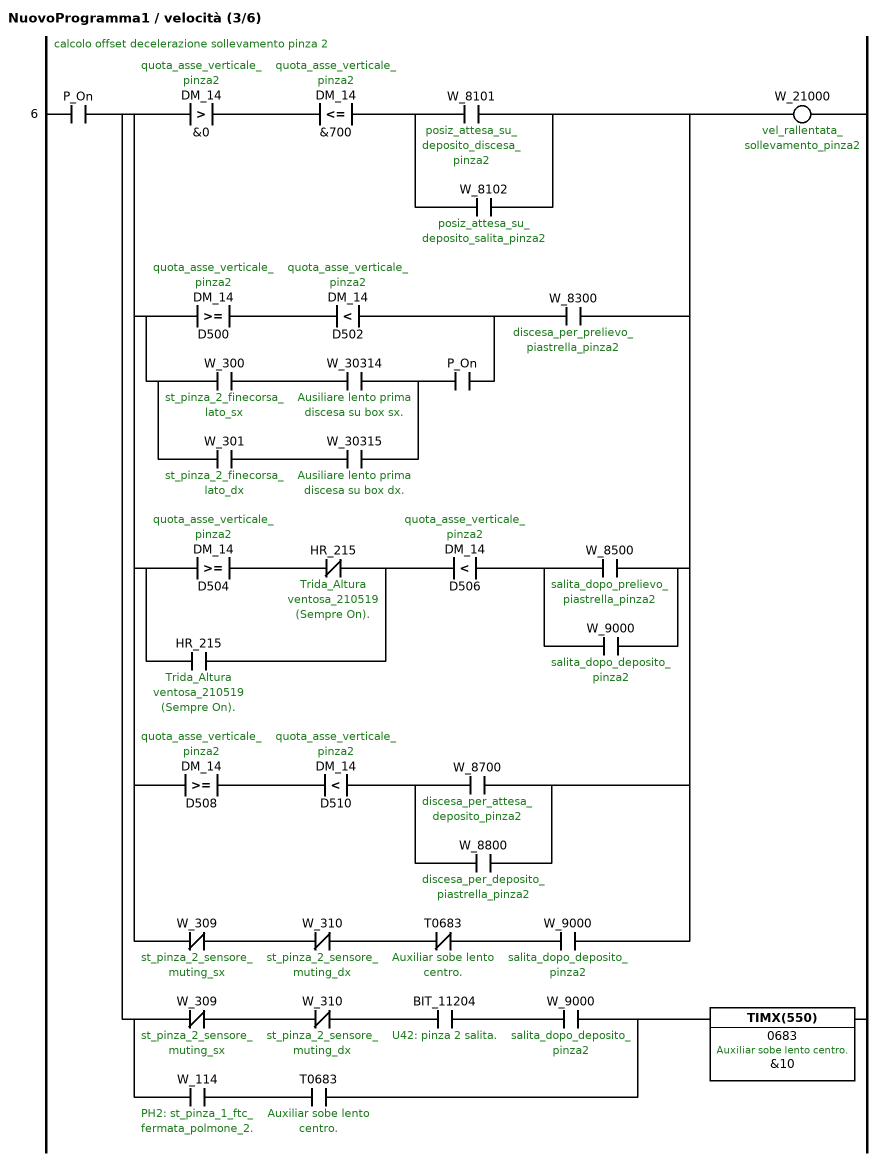
; [picture p120: NuovoProgramma1 / velocità, rungs 6-6]
; rung 6: calcolo offset decelerazione sollevamento pinza 2
LD P_On
OUT TR0
LD>SL(323) DM_14 &0  ; quota_asse_verticale_pinza2
AND<=SL(318) DM_14 &700  ; quota_asse_verticale_pinza2
LD W_8101  ; posiz_attesa_su_deposito_discesa_pinza2
OR W_8102  ; posiz_attesa_su_deposito_salita_pinza2
ANDLD
LD>=SL(328) DM_14 D500  ; quota_asse_verticale_pinza2
AND<SL(313) DM_14 D502  ; quota_asse_verticale_pinza2
LD W_300  ; st_pinza_2_finecorsa_lato_sx
AND W_30314  ; Ausiliare lento prima discesa su box sx.
LD W_301  ; st_pinza_2_finecorsa_lato_dx
AND W_30315  ; Ausiliare lento prima discesa su box dx.
ORLD
AND P_On
ORLD
AND W_8300  ; discesa_per_prelievo_piastrella_pinza2
ORLD
LD>=SL(328) DM_14 D504  ; quota_asse_verticale_pinza2
ANDNOT HR_215  ; Trida_Altura ventosa_210519 (Sempre On).  // HR 2.15: Ventosa voltava a entrar veloz pouco antes de para no alto. / .
OR HR_215  ; Trida_Altura ventosa_210519 (Sempre On).  // HR 2.15: Ventosa voltava a entrar veloz pouco antes de para no alto. / .
AND<SL(313) DM_14 D506  ; quota_asse_verticale_pinza2
LD W_8500  ; salita_dopo_prelievo_piastrella_pinza2
OR W_9000  ; salita_dopo_deposito_pinza2
ANDLD
ORLD
LD>=SL(328) DM_14 D508  ; quota_asse_verticale_pinza2
AND<SL(313) DM_14 D510  ; quota_asse_verticale_pinza2
LD W_8700  ; discesa_per_attesa_deposito_pinza2
OR W_8800  ; discesa_per_deposito_piastrella_pinza2
ANDLD
ORLD
LDNOT W_309  ; st_pinza_2_sensore_muting_sx  // Pinça no centro. / .
ANDNOT W_310  ; st_pinza_2_sensore_muting_dx  // Pinça no centro. / .
ANDNOT T0683  ; Auxiliar sobe lento centro.
AND W_9000  ; salita_dopo_deposito_pinza2
ORLD
ANDLD
OUT W_21000  ; vel_rallentata_sollevamento_pinza2
LD TR0
LDNOT W_309  ; st_pinza_2_sensore_muting_sx  // Pinça no centro. / .
ANDNOT W_310  ; st_pinza_2_sensore_muting_dx  // Pinça no centro. / .
AND BIT_11204  ; U42: pinza 2 salita.
AND W_9000  ; salita_dopo_deposito_pinza2
LD W_114  ; PH2: st_pinza_1_ftc_fermata_polmone_2.
AND T0683  ; Auxiliar sobe lento centro.  // Auto-alimento para efetuar controle de velocidade somente no 1º plano depositado. / .
ORLD
ANDLD
TIMX(550) 0683 &10  ; Auxiliar sobe lento centro.  // Auxiliar início sobe lento centro. / "Puxa" as peças do 1º plano depositado. / .

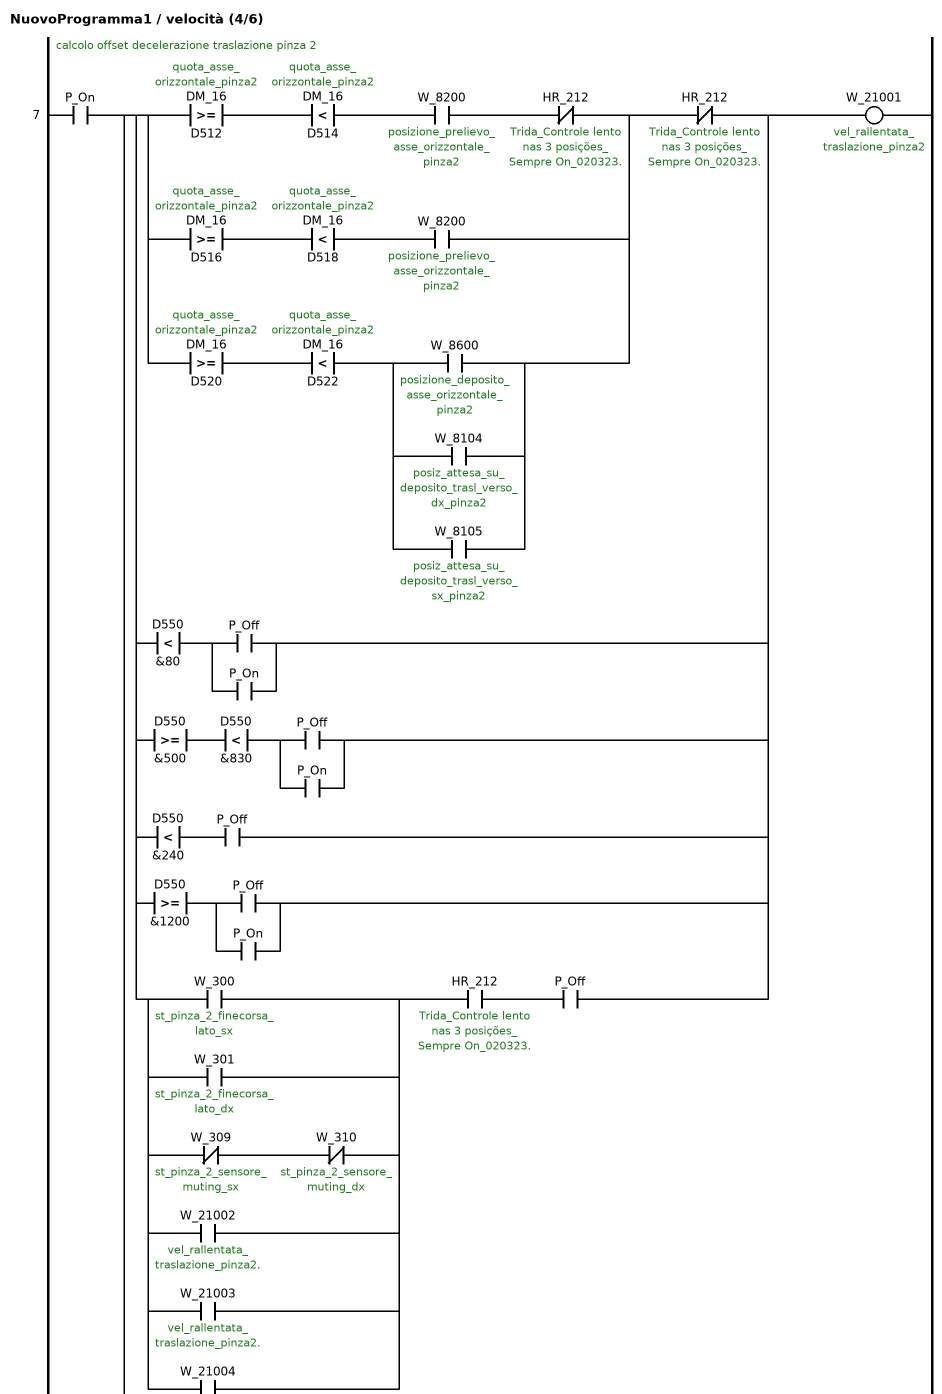

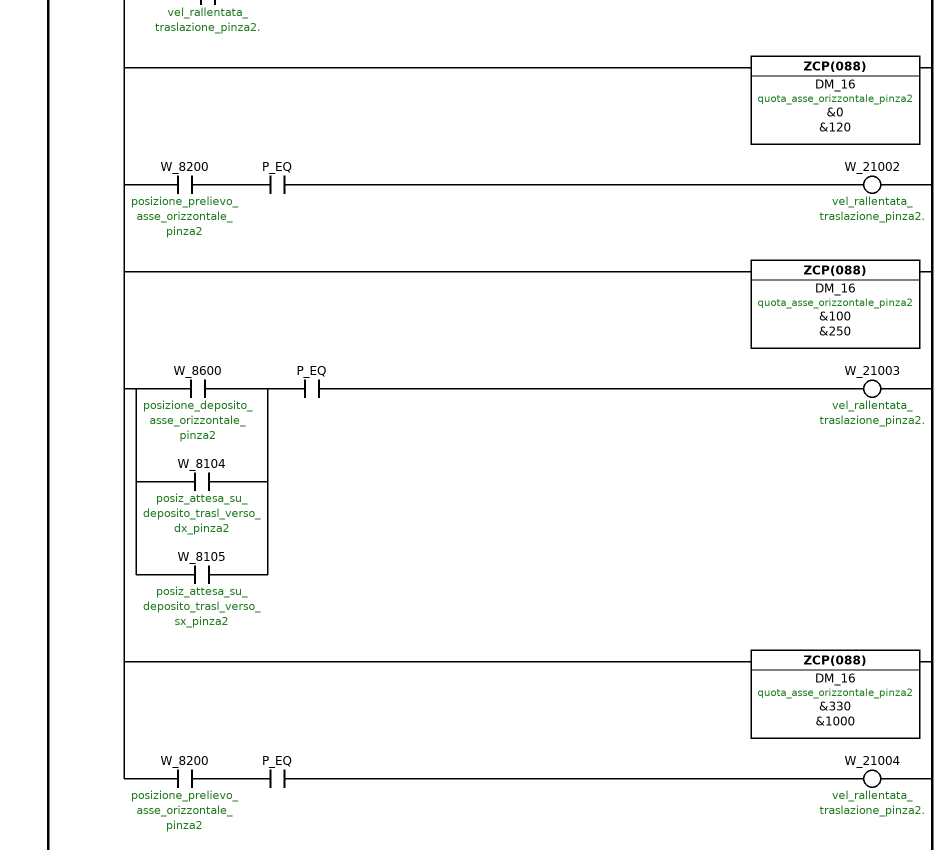
; rung 7: calcolo offset decelerazione traslazione pinza 2
LD P_On
OUT TR0
LD>=SL(328) DM_16 D512  ; quota_asse_orizzontale_pinza2
AND<SL(313) DM_16 D514  ; quota_asse_orizzontale_pinza2
AND W_8200  ; posizione_prelievo_asse_orizzontale_pinza2
ANDNOT HR_212  ; Trida_Controle lento nas 3 posições_Sempre On_020323.
LD>=SL(328) DM_16 D516  ; quota_asse_orizzontale_pinza2
AND<SL(313) DM_16 D518  ; quota_asse_orizzontale_pinza2
AND W_8200  ; posizione_prelievo_asse_orizzontale_pinza2
ORLD
LD>=SL(328) DM_16 D520  ; quota_asse_orizzontale_pinza2
AND<SL(313) DM_16 D522  ; quota_asse_orizzontale_pinza2
LD W_8600  ; posizione_deposito_asse_orizzontale_pinza2
OR W_8104  ; posiz_attesa_su_deposito_trasl_verso_dx_pinza2
OR W_8105  ; posiz_attesa_su_deposito_trasl_verso_sx_pinza2
ANDLD
ORLD
ANDNOT HR_212  ; Trida_Controle lento nas 3 posições_Sempre On_020323.
LD<SL(313) D550 &80
LD P_Off
OR P_On
ANDLD
ORLD
LD>=SL(328) D550 &500
AND<SL(313) D550 &830
LD P_Off
OR P_On
ANDLD
ORLD
LD<SL(313) D550 &240
AND P_Off
ORLD
LD>=SL(328) D550 &1200
LD P_Off
OR P_On
ANDLD
ORLD
LD W_300  ; st_pinza_2_finecorsa_lato_sx  // Pinça à esquerda. / .
OR W_301  ; st_pinza_2_finecorsa_lato_dx  // Pinça à direita. / .
LDNOT W_309  ; st_pinza_2_sensore_muting_sx  // Pinça no centro. / .
ANDNOT W_310  ; st_pinza_2_sensore_muting_dx  // Pinça no centro. / .
ORLD
OR W_21002  ; vel_rallentata_traslazione_pinza2.
OR W_21003  ; vel_rallentata_traslazione_pinza2.
OR W_21004  ; vel_rallentata_traslazione_pinza2.
AND HR_212  ; Trida_Controle lento nas 3 posições_Sempre On_020323.
AND P_Off
ORLD
ANDLD
OUT W_21001  ; vel_rallentata_traslazione_pinza2
LD TR0
ZCP(088) DM_16 &0 &120  ; quota_asse_orizzontale_pinza2  // Valor contagem na esquerda: 0. / .
AND W_8200  ; posizione_prelievo_asse_orizzontale_pinza2
AND P_EQ
OUT W_21002  ; vel_rallentata_traslazione_pinza2.
LD TR0
ZCP(088) DM_16 &100 &250  ; quota_asse_orizzontale_pinza2  // Valor contagem no centro: +/- 220. / .
LD W_8600  ; posizione_deposito_asse_orizzontale_pinza2
OR W_8104  ; posiz_attesa_su_deposito_trasl_verso_dx_pinza2
OR W_8105  ; posiz_attesa_su_deposito_trasl_verso_sx_pinza2
ANDLD
AND P_EQ
OUT W_21003  ; vel_rallentata_traslazione_pinza2.
LD TR0
ZCP(088) DM_16 &330 &1000  ; quota_asse_orizzontale_pinza2  // Valor contagem na direita: +/- 360. / .
AND W_8200  ; posizione_prelievo_asse_orizzontale_pinza2
AND P_EQ
OUT W_21004  ; vel_rallentata_traslazione_pinza2.

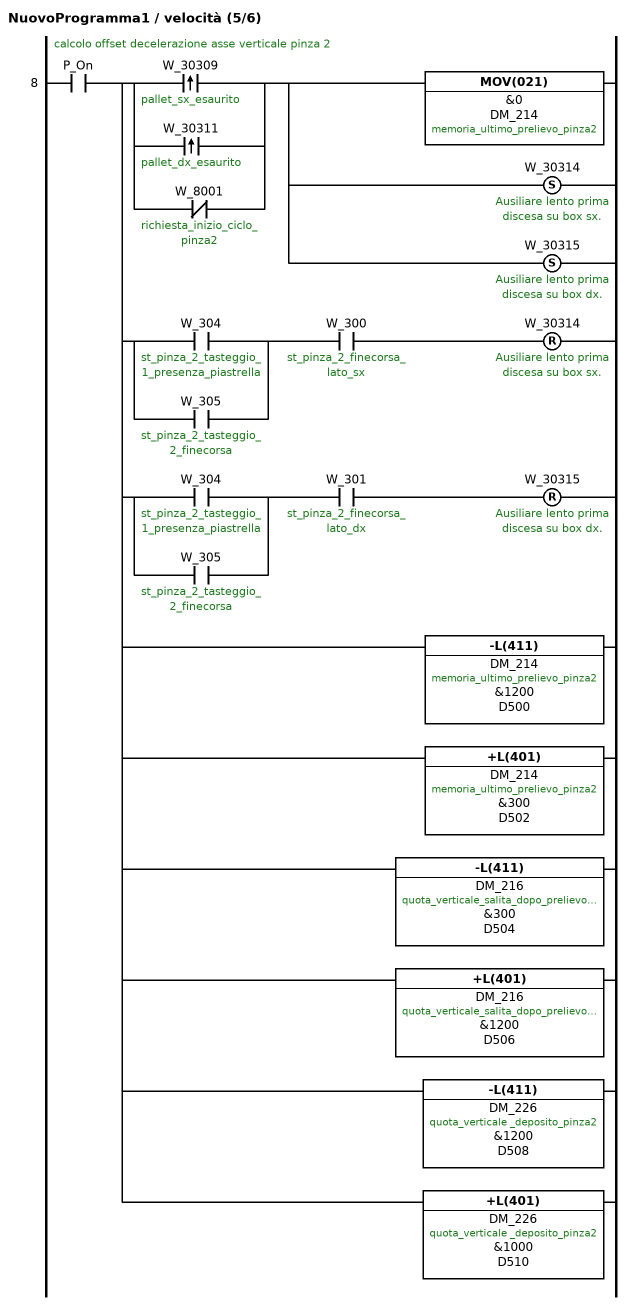
; rung 8: calcolo offset decelerazione asse verticale pinza 2
LD P_On
OUT TR0
@LD W_30309  ; pallet_sx_esaurito
@OR W_30311  ; pallet_dx_esaurito
ORNOT W_8001  ; richiesta_inizio_ciclo_pinza2
ANDLD
MOV(021) &0 DM_214  ; memoria_ultimo_prelievo_pinza2
SET W_30314  ; Ausiliare lento prima discesa su box sx.
SET W_30315  ; Ausiliare lento prima discesa su box dx.
LD TR0
LD W_304  ; st_pinza_2_tasteggio_1_presenza_piastrella
OR W_305  ; st_pinza_2_tasteggio_2_finecorsa
ANDLD
AND W_300  ; st_pinza_2_finecorsa_lato_sx
RSET W_30314  ; Ausiliare lento prima discesa su box sx.
LD TR0
LD W_304  ; st_pinza_2_tasteggio_1_presenza_piastrella
OR W_305  ; st_pinza_2_tasteggio_2_finecorsa
ANDLD
AND W_301  ; st_pinza_2_finecorsa_lato_dx
RSET W_30315  ; Ausiliare lento prima discesa su box dx.
LD TR0
-L(411) DM_214 &1200 D500  ; memoria_ultimo_prelievo_pinza2
+L(401) DM_214 &300 D502  ; memoria_ultimo_prelievo_pinza2
-L(411) DM_216 &300 D504  ; quota_verticale_salita_dopo_prelievo_pinza2
+L(401) DM_216 &1200 D506  ; quota_verticale_salita_dopo_prelievo_pinza2
-L(411) DM_226 &1200 D508  ; quota_verticale _deposito_pinza2
+L(401) DM_226 &1000 D510  ; quota_verticale _deposito_pinza2

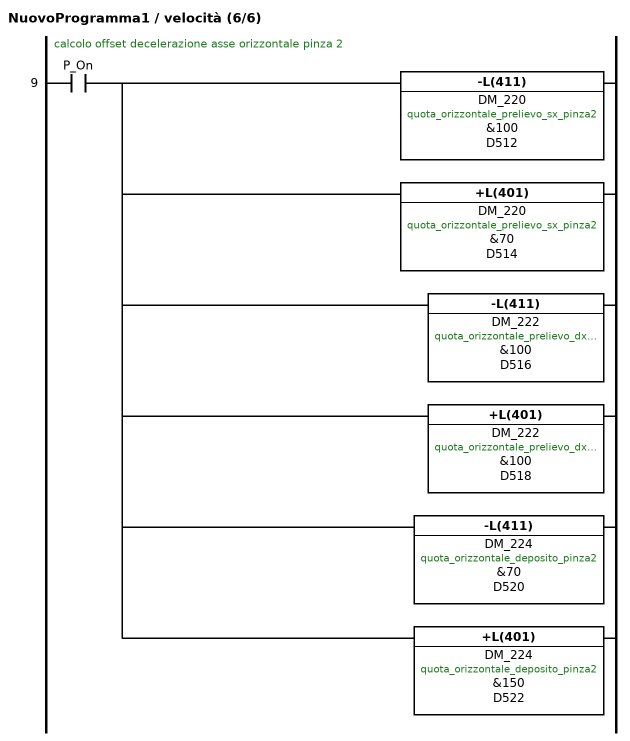
; rung 9: calcolo offset decelerazione asse orizzontale pinza 2
LD P_On
-L(411) DM_220 &100 D512  ; quota_orizzontale_prelievo_sx_pinza2
+L(401) DM_220 &70 D514  ; quota_orizzontale_prelievo_sx_pinza2
-L(411) DM_222 &100 D516  ; quota_orizzontale_prelievo_dx_pinza2
+L(401) DM_222 &100 D518  ; quota_orizzontale_prelievo_dx_pinza2
-L(411) DM_224 &70 D520  ; quota_orizzontale_deposito_pinza2
+L(401) DM_224 &150 D522  ; quota_orizzontale_deposito_pinza2

### Section END
; rung 0
END(001)

## Program NuovoProgramma2 (interrupt task 140)

### Section Sezione1

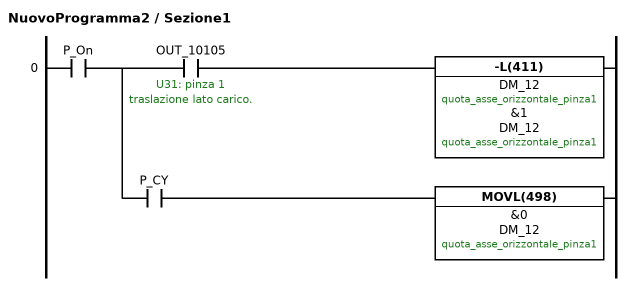
; rung 0
LD P_On
OUT TR0
AND OUT_10105  ; U31: pinza 1 traslazione lato carico.
-L(411) DM_12 &1 DM_12  ; quota_asse_orizzontale_pinza1
LD TR0
AND P_CY
MOVL(498) &0 DM_12  ; quota_asse_orizzontale_pinza1

### Section END
; rung 0
END(001)

## Program NuovoProgramma3 (interrupt task 141)

### Section Sezione1

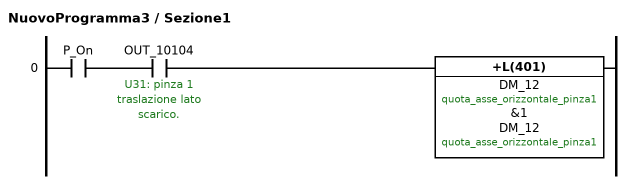
; rung 0
LD P_On
AND OUT_10104  ; U31: pinza 1 traslazione lato scarico.
+L(401) DM_12 &1 DM_12  ; quota_asse_orizzontale_pinza1

### Section END
; rung 0
END(001)

## Program NuovoProgramma4 (interrupt task 142)

### Section Sezione1

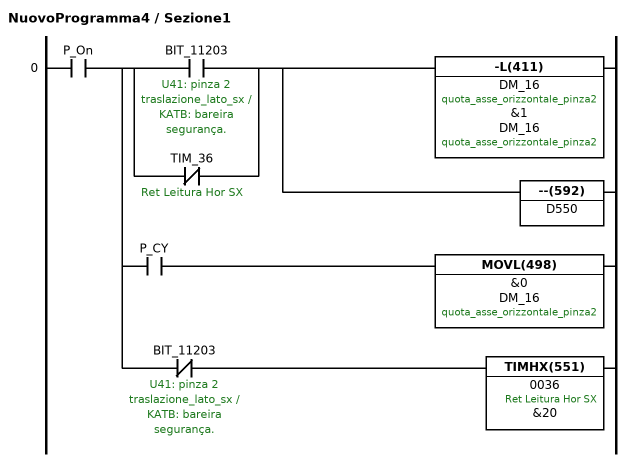
; rung 0
LD P_On
OUT TR0
LD BIT_11203  ; U41: pinza 2 traslazione_lato_sx / KATB: bareira segurança.
ORNOT TIM_36  ; Ret Leitura Hor SX
ANDLD
-L(411) DM_16 &1 DM_16  ; quota_asse_orizzontale_pinza2
--(592) D550
LD TR0
AND P_CY
MOVL(498) &0 DM_16  ; quota_asse_orizzontale_pinza2
LD TR0
ANDNOT BIT_11203  ; U41: pinza 2 traslazione_lato_sx / KATB: bareira segurança.
TIMHX(551) 0036 &20  ; Ret Leitura Hor SX

### Section END
; rung 0
END(001)

## Program NuovoProgramma5 (interrupt task 143)

### Section Sezione1

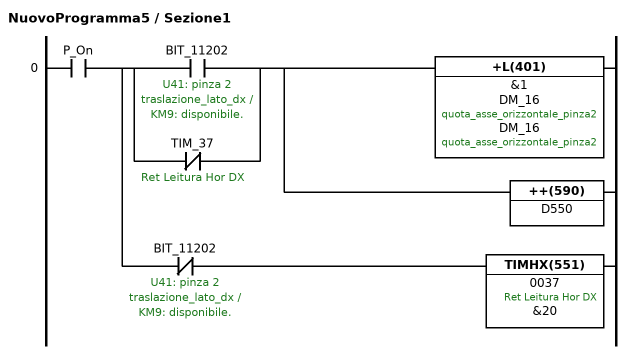
; rung 0
LD P_On
OUT TR0
LD BIT_11202  ; U41: pinza 2 traslazione_lato_dx / KM9: disponibile.
ORNOT TIM_37  ; Ret Leitura Hor DX
ANDLD
+L(401) &1 DM_16 DM_16  ; quota_asse_orizzontale_pinza2
++(590) D550
LD TR0
ANDNOT BIT_11202  ; U41: pinza 2 traslazione_lato_dx / KM9: disponibile.
TIMHX(551) 0037 &20  ; Ret Leitura Hor DX

### Section END
; rung 0
END(001)

## Function block Modbus_Write_Parameter
VAR_INPUT
  Unit_n : INT;
  Serial_port_n : INT;
  Node : INT;
  Parameter : WORD;
  Value : WORD;
  start_comm : BOOL;
END_VAR
VAR_OUTPUT
  Busy : BOOL;
  Comms_error : BOOL;
  Error_Code : WORD;
END_VAR
VAR
  source : ARRAY[0..5] OF WORD;  (* Source area of the CMND *)
  control : ARRAY[0..5] OF WORD;  (* Control Data for the CMND instruction *)
  response : ARRAY[0..4] OF WORD;  (* Response area of the CMND istruction *)
  comm : BOOL;  (* Communication enabled *)
  stop_comm : BOOL;  (* Stops the communication *)
  tmp : DINT;  (* Temporary data for math *)
  port_n AT A218 : WORD;  (* Communication port number assigned with automatic allocation *)
  used_port : WORD;  (* Current communication port *)
  stby : BOOL;  (* Delays the reading of the status for one scan after comms activation *)
  First_Cycle_after_Network_Comms AT A214 : WORD;  (* Turns On on the first scan right after the completion of the communication function *)
  Fisrt_Cycle_after_Comms_Error AT A215 : WORD;  (* Turns On during the first scan after a communication error *)
  error_code_storage_location AT A216 : DWORD;  (* Returns the memory address where the error code is stored *)
  tmp_ir0 : DWORD;  (* Stores the content of IR0 *)
  actual_error_code_ptr : DWORD;  (* Points to the memory location that contains the error code *)
END_VAR

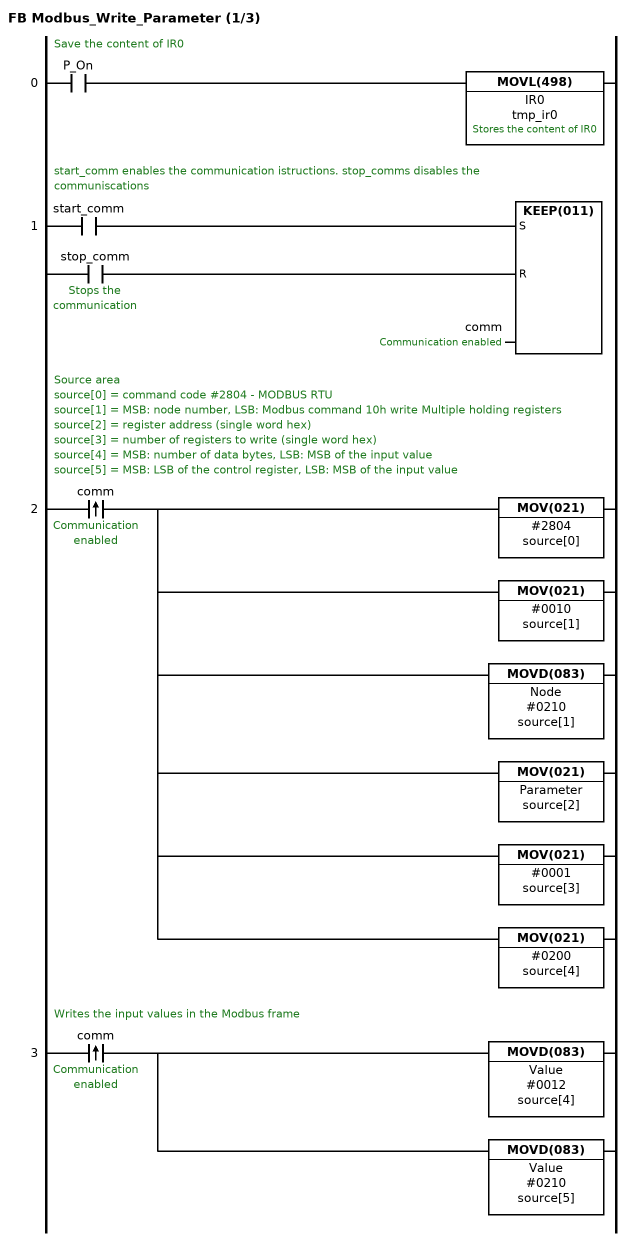
; rung 0: Save the content of IR0
LD P_On
MOVL(498) IR0 tmp_ir0  ; Stores the content of IR0
; rung 1: start_comm enables the communication istructions. stop_comms disables the communiscations
LD start_comm
LD stop_comm  ; Stops the communication
KEEP(011) comm  ; Communication enabled
; rung 2: Source area / source[0] = command code #2804 - MODBUS RTU / source[1] = MSB: node number, LSB: Modbus command 10h write Multiple holding registers / source[2] = register address (single word hex) / source[3] = number of registers to write (single word hex) / source[4] = MSB: number of data bytes, LSB: MSB of the input value / source[5] = MSB: LSB of the control register, LSB: MSB of the input value
@LD comm  ; Communication enabled
MOV(021) #2804 source[0]
MOV(021) #0010 source[1]
MOVD(083) Node #0210 source[1]
MOV(021) Parameter source[2]
MOV(021) #0001 source[3]
MOV(021) #0200 source[4]
; rung 3: Writes the input values in the Modbus frame
@LD comm  ; Communication enabled
MOVD(083) Value #0012 source[4]
MOVD(083) Value #0210 source[5]

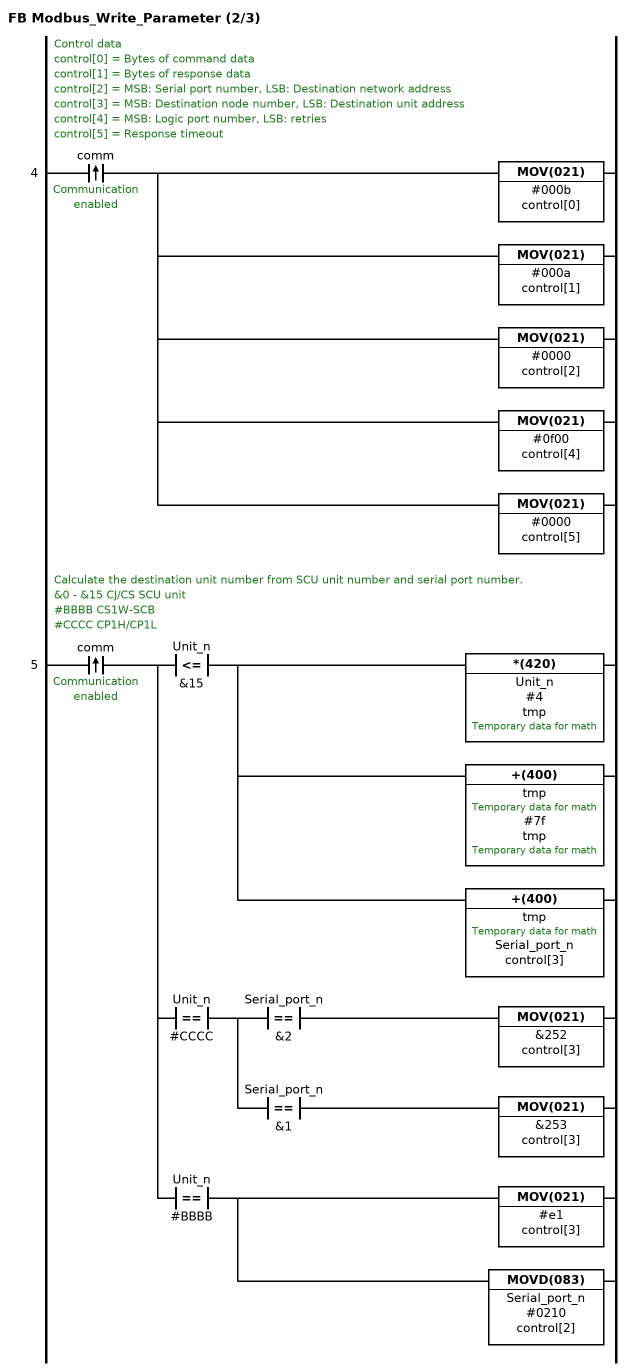
; rung 4: Control data / control[0] = Bytes of command data / control[1] = Bytes of response data / control[2] = MSB: Serial port number, LSB: Destination network address / control[3] = MSB: Destination node number, LSB: Destination unit address / control[4] = MSB: Logic port number, LSB: retries / control[5] = Response timeout
@LD comm  ; Communication enabled
MOV(021) #000b control[0]
MOV(021) #000a control[1]
MOV(021) #0000 control[2]
MOV(021) #0f00 control[4]
MOV(021) #0000 control[5]
; rung 5: Calculate the destination unit number from SCU unit number and serial port number. / &0 - &15 CJ/CS SCU unit / #BBBB CS1W-SCB / #CCCC CP1H/CP1L
@LD comm  ; Communication enabled
OUT TR0
AND<=(315) Unit_n &15
*(420) Unit_n #4 tmp  ; Temporary data for math
+(400) tmp #7f tmp  ; Temporary data for math
+(400) tmp Serial_port_n control[3]  ; Temporary data for math
LD TR0
AND=(300) Unit_n #CCCC
OUT TR1
AND=(300) Serial_port_n &2
MOV(021) &252 control[3]
LD TR1
AND=(300) Serial_port_n &1
MOV(021) &253 control[3]
LD TR0
AND=(300) Unit_n #BBBB
MOV(021) #e1 control[3]
MOVD(083) Serial_port_n #0210 control[2]

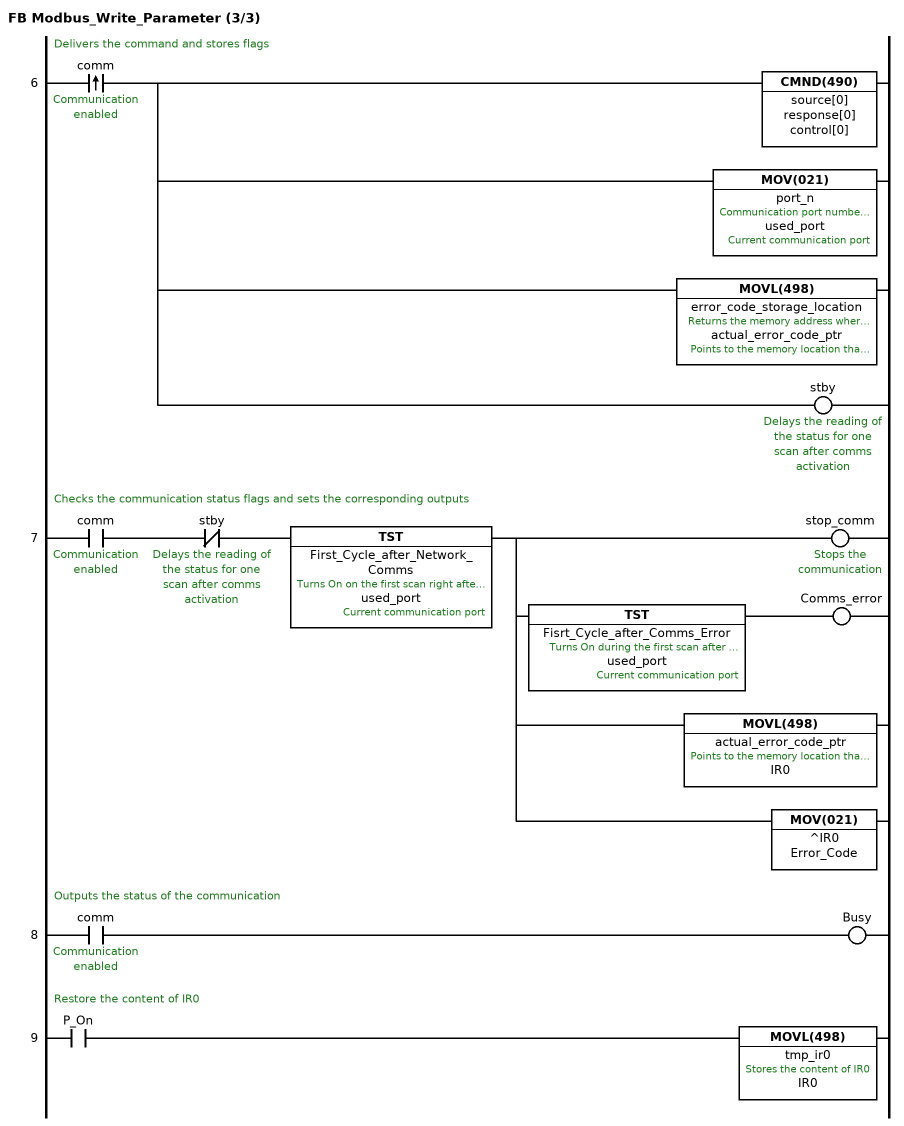
; rung 6: Delivers the command and stores flags
@LD comm  ; Communication enabled
CMND(490) source[0] response[0] control[0]
MOV(021) port_n used_port  ; Communication port number assigned with automatic allocation, Current communication port
MOVL(498) error_code_storage_location actual_error_code_ptr  ; Returns the memory address where the error code is stored, Points to the memory location that contains the error code
OUT stby  ; Delays the reading of the status for one scan after comms activation
; rung 7: Checks the communication status flags and sets the corresponding outputs
LD comm  ; Communication enabled
ANDNOT stby  ; Delays the reading of the status for one scan after comms activation
ANDTST(350) First_Cycle_after_Network_Comms used_port  ; Turns On on the first scan right after the completion of the communication function, Current communication port
OUT TR0
OUT stop_comm  ; Stops the communication
ANDTST(350) Fisrt_Cycle_after_Comms_Error used_port  ; Turns On during the first scan after a communication error, Current communication port
OUT Comms_error
LD TR0
MOVL(498) actual_error_code_ptr IR0  ; Points to the memory location that contains the error code
MOV(021) ^IR0 Error_Code
; rung 8: Outputs the status of the communication
LD comm  ; Communication enabled
OUT Busy
; rung 9: Restore the content of IR0
LD P_On
MOVL(498) tmp_ir0 IR0  ; Stores the content of IR0